FUNCTION_BLOCK FB_KvFeedForward

// BOOL:  True / False
// LREAL: Long real decimal number
 
// Input variables
VAR_INPUT
    bEnable         : BOOL;         // Enable signal for KvFF
    fXDotref        : LREAL;     	// Velocity reference [m/s]
    fPa             : LREAL;        // Pressure piston side [bar]
    fPb             : LREAL;        // Pressure rod side [bar]
    fPs             : LREAL;        // Supply pressure [bar]
    fA              : LREAL;        // Piston area [m^2]
    fAr             : LREAL;        // Rod side area [m^2]
END_VAR
 
// Output variables
VAR_OUTPUT
    fU_FF           : LREAL;        // Feed-forward valve command [-1, 1]
    fKv             : LREAL;        // Calculated Kv [L/min / bar^0.5]
    fFlow           : LREAL;        // Required flow [L/min]
    fdP             : LREAL;        // Active pressure drop [bar]
END_VAR
 
// Variables
VAR
    fSpoolPos       : LREAL;        // Spool position from polynomial [-1, 1]
    fKv_min         : LREAL := 0.1; // Minimum Kv for polynomial validity
	fSpoolPosCtrl   : LREAL;        
END_VAR

// Feed forward based on calculated Kv with polynomial spool compensation.

IF NOT bEnable THEN
    fU_FF    := 0.0;
    fKv      := 0.0;
    fFlow    := 0.0;
    fdP      := 0.0;
 
ELSIF fXDotref > 0.0 THEN                                       // Cylinder moving up
    fFlow   := fXDotref * fA * 60000.0;                         // Required flow [L/min]
    fdP     := fPs - fPa;                                      	// Pressure drop [bar]
 
    IF fdP <= 0.0 THEN                                         	// Avoiding division by zero
        fKv := 4.0;
    ELSE
        fKv := ABS(fFlow) / SQRT(fdP);                         	// Calculates Kv [L/min / bar^0.5]
    END_IF
 
    IF fKv >= fKv_min THEN									 	// Upwards motion spool polynomial
//         fSpoolPos :=  -0.00038291 * EXPT(fKv, 6)
//                       -0.0083821  * EXPT(fKv, 5)
//                       +0.11362    * EXPT(fKv, 4)
//                       -0.44825    * EXPT(fKv, 3)
//                       +0.64863    * EXPT(fKv, 2)
//                       +0.019414   * fKv
//                       +0.25505;
					  
		fSpoolPos :=  +0.0018653  * EXPT(fKv, 6)
              -0.033672    * EXPT(fKv, 5)
              +0.22033     * EXPT(fKv, 4)
              -0.65618     * EXPT(fKv, 3)
              +0.83411     * EXPT(fKv, 2)
              -0.047269    * fKv
              +0.26252;
					   		
	 
    ELSE
		//fSpoolPos := 0.236 + 0.270407 * fKv;   					// Linear approximation for low Kv
		fSpoolPos := 0.231 + 0.270407 * fKv;   						// Linear approximation for low Kv
    END_IF
	//fSpoolPosCtrl := 1.1182 * fSpoolPos - 0.0325;			// Original
	fSpoolPosCtrl := (fSpoolPos + 0.0325) / 1.1182;	
    fU_FF := LIMIT(-1.0, -fSpoolPosCtrl, 1.0);		
                     	
 
ELSIF fXDotref < 0.0 THEN                                       // Cylinder going down
    fFlow   := fXDotref * fAr * 60000.0;                        // Required flow [L/min]
    fdP     := fPs - fPb;                                       // Pressure drop [bar]
 
    IF fdP <= 0.0 THEN                                          // Avoiding division by zero
        fKv := 4.0;
    ELSE
        fKv := ABS(fFlow) / SQRT(fdP);                         	// Calculates Kv [L/min / bar^0.5]
    END_IF
 
    IF fKv >= fKv_min THEN										// Downwards motion spool polynomial
//         fSpoolPos :=  0.001656  * EXPT(fKv, 6)
//                       -0.026792 * EXPT(fKv, 5)
//                       +0.16458  * EXPT(fKv, 4)
//                       -0.46999  * EXPT(fKv, 3)
//                       +0.56415  * EXPT(fKv, 2)
//                       +0.08632  * fKv
//                       +0.22422;
					  
		fSpoolPos :=  +0.00098272 * EXPT(fKv, 6)
              -0.017507    * EXPT(fKv, 5)
              +0.11599     * EXPT(fKv, 4)
              -0.34851     * EXPT(fKv, 3)
              +0.41222     * EXPT(fKv, 2)
              +0.17643     * fKv
              +0.2076;  
					
    ELSE
		//fSpoolPos := 0.215 + 0.230397 * fKv;   					// Linear from deadband to polynomial
		fSpoolPos := 0.1865 + 0.230397 * fKv;   					// Linear from deadband to polynomial
		// change from 0.1965
    END_IF
		//fSpoolPosCtrl := 1.1075 * fSpoolPos - 0.0416;		// Original 
		fSpoolPosCtrl := (fSpoolPos + 0.0416) / 1.1075;
    	fU_FF := LIMIT(-1.0, fSpoolPosCtrl, 1.0);		                      	
 
ELSE
    fU_FF    := 0.0;
    fKv      := 0.0;
    fFlow    := 0.0;
    fdP      := 0.0;
 
END_IF

END_FUNCTION_BLOCK

(* stored: Version 1.1.0.1
   POU FB_KvFeedForward: Id {0481b253-c5ae-423c-9bd3-30b2fe072313}, SpecialFunc None *)
